PROGRAM MAIN
VAR
END_VAR

onOffLed();
byteCounter();
sevenSegProg();

END_PROGRAM

(* stored: Version 1.1.0.1, ProductVersion 3.1.4024.5
   POU MAIN: Id {167442c7-625b-4f99-be1c-db4574452fd9}, SpecialFunc None *)
